INTERFACE I_Serializer EXTENDS I_Disposable

METHOD PUBLIC AddBase64 : I_Serializer
VAR_INPUT
	pBytes : POINTER TO BYTE;
	nBytes : DINT;
END_VAR
END_METHOD

METHOD PUBLIC AddBool : I_Serializer
VAR_INPUT
	Value : BOOL;
END_VAR
END_METHOD

METHOD PUBLIC AddByte : I_Serializer
VAR_INPUT
	Value : BYTE;
END_VAR
END_METHOD

METHOD PUBLIC AddBytesAsHex : I_Serializer
VAR_INPUT
	pBytes : POINTER TO BYTE;
	nBytes : DINT;
END_VAR
END_METHOD

METHOD PUBLIC AddDateTime : I_Serializer
VAR_INPUT
	Value : DATE_AND_TIME;
END_VAR
END_METHOD

METHOD PUBLIC AddDcTime : I_Serializer
VAR_INPUT
	Value : DCTIME;
END_VAR
END_METHOD

METHOD PUBLIC AddDint : I_Serializer
VAR_INPUT
	Value : DINT;
END_VAR
END_METHOD

METHOD PUBLIC AddDword : I_Serializer
VAR_INPUT
	Value : DWORD;
END_VAR
END_METHOD

METHOD PUBLIC AddFileTime : I_Serializer
VAR_INPUT
	Value : FILETIME;
END_VAR
END_METHOD

METHOD PUBLIC AddInt : I_Serializer
VAR_INPUT
	Value : INT;
END_VAR
END_METHOD

METHOD PUBLIC AddKey : I_Serializer
VAR_INPUT
	Key : T_MAXSTRING;
END_VAR
END_METHOD

METHOD PUBLIC AddKeyBase64 : I_Serializer
VAR_INPUT
	Key : T_MAXSTRING;
	pBytes : POINTER TO BYTE;
	nBytes : DINT;
END_VAR
END_METHOD

METHOD PUBLIC AddKeyBool : I_Serializer
VAR_INPUT
	Key : T_MAXSTRING;
	Value : BOOL;
END_VAR
END_METHOD

METHOD PUBLIC AddKeyByte : I_Serializer
VAR_INPUT
	Key : T_MAXSTRING;
	Value : BYTE;
END_VAR
END_METHOD

METHOD PUBLIC AddKeyBytesAsHex : I_Serializer
VAR_INPUT
	Key : T_MAXSTRING;
	pBytes : POINTER TO BYTE;
	nBytes : DINT;
END_VAR
END_METHOD

METHOD PUBLIC AddKeyDateTime : I_Serializer
VAR_INPUT
	Key : T_MAXSTRING;
	Value : DATE_AND_TIME;
END_VAR
END_METHOD

METHOD PUBLIC AddKeyDcTime : I_Serializer
VAR_INPUT
	Key : T_MAXSTRING;
	Value : DCTIME;
END_VAR
END_METHOD

METHOD PUBLIC AddKeyDint : I_Serializer
VAR_INPUT
	Key : T_MAXSTRING;
	Value : DINT;
END_VAR
END_METHOD

METHOD PUBLIC AddKeyDword : I_Serializer
VAR_INPUT
	Key : T_MAXSTRING;
	Value : DWORD;
END_VAR
END_METHOD

METHOD PUBLIC AddKeyFileTime : I_Serializer
VAR_INPUT
	Key : T_MAXSTRING;
	Value : FILETIME;
END_VAR
END_METHOD

METHOD PUBLIC AddKeyInt : I_Serializer
VAR_INPUT
	Key : T_MAXSTRING;
	Value : INT;
END_VAR
END_METHOD

METHOD PUBLIC AddKeyLint : I_Serializer
VAR_INPUT
	Key : T_MAXSTRING;
	Value : LINT;
END_VAR
END_METHOD

METHOD PUBLIC AddKeyLreal : I_Serializer
VAR_INPUT
	Key : T_MAXSTRING;
	Value : LREAL;
END_VAR
END_METHOD

METHOD PUBLIC AddKeyLtime : I_Serializer
VAR_INPUT
	Key : T_MAXSTRING;
	Value : LTIME;
END_VAR
END_METHOD

METHOD PUBLIC AddKeyLword : I_Serializer
VAR_INPUT
	Key : T_MAXSTRING;
	Value : LWORD;
END_VAR
END_METHOD

METHOD PUBLIC AddKeyNull : I_Serializer
VAR_INPUT
	Key : T_MAXSTRING;
END_VAR
END_METHOD

METHOD PUBLIC AddKeyReal : I_Serializer
VAR_INPUT
	Key : T_MAXSTRING;
	Value : REAL;
END_VAR
END_METHOD

METHOD PUBLIC AddKeySint : I_Serializer
VAR_INPUT
	Key : T_MAXSTRING;
	Value : SINT;
END_VAR
END_METHOD

METHOD PUBLIC AddKeyString : I_Serializer
VAR_INPUT
	Key : T_MAXSTRING;
	Value : T_MAXSTRING;
END_VAR
END_METHOD

METHOD PUBLIC AddKeyStringByRef : I_Serializer
VAR_INPUT
	Key : T_MAXSTRING;
	Value : REFERENCE TO STRING;
END_VAR
END_METHOD

METHOD PUBLIC AddKeyTime : I_Serializer
VAR_INPUT
	Key : T_MAXSTRING;
	Value : TIME;
END_VAR
END_METHOD

METHOD PUBLIC AddKeyTod : I_Serializer
VAR_INPUT
	Key : T_MAXSTRING;
	Value : TOD;
END_VAR
END_METHOD

METHOD PUBLIC AddKeyUdint : I_Serializer
VAR_INPUT
	Key : T_MAXSTRING;
	Value : UDINT;
END_VAR
END_METHOD

METHOD PUBLIC AddKeyUint : I_Serializer
VAR_INPUT
	Key : T_MAXSTRING;
	Value : UINT;
END_VAR
END_METHOD

METHOD PUBLIC AddKeyUlint : I_Serializer
VAR_INPUT
	Key : T_MAXSTRING;
	Value : ULINT;
END_VAR
END_METHOD

METHOD PUBLIC AddKeyUsint : I_Serializer
VAR_INPUT
	Key : T_MAXSTRING;
	Value : USINT;
END_VAR
END_METHOD

METHOD PUBLIC AddKeyWord : I_Serializer
VAR_INPUT
	Key : T_MAXSTRING;
	Value : WORD;
END_VAR
END_METHOD

METHOD PUBLIC AddLint : I_Serializer
VAR_INPUT
	Value : LINT;
END_VAR
END_METHOD

METHOD PUBLIC AddLreal : I_Serializer
VAR_INPUT
	Value : LREAL;
END_VAR
END_METHOD

METHOD PUBLIC AddLtime : I_Serializer
VAR_INPUT
	Value : LTIME;
END_VAR
END_METHOD

METHOD PUBLIC AddLword : I_Serializer
VAR_INPUT
	Value : LWORD;
END_VAR
END_METHOD

METHOD PUBLIC AddNull : I_Serializer
VAR_INPUT
END_VAR
END_METHOD

METHOD PUBLIC AddReal : I_Serializer
VAR_INPUT
	Value : REAL;
END_VAR
END_METHOD

METHOD PUBLIC AddSint : I_Serializer
VAR_INPUT
	Value : SINT;
END_VAR
END_METHOD

METHOD PUBLIC AddString : I_Serializer
VAR_INPUT
	Value : T_MAXSTRING;
END_VAR
END_METHOD

METHOD PUBLIC AddStringByRef : I_Serializer
VAR_INPUT
	Value : REFERENCE TO STRING;
END_VAR
END_METHOD

METHOD PUBLIC AddTime : I_Serializer
VAR_INPUT
	Value : TIME;
END_VAR
END_METHOD

METHOD PUBLIC AddTod : I_Serializer
VAR_INPUT
	Value : TOD;
END_VAR
END_METHOD

METHOD PUBLIC AddUdint : I_Serializer
VAR_INPUT
	Value : UDINT;
END_VAR
END_METHOD

METHOD PUBLIC AddUint : I_Serializer
VAR_INPUT
	Value : UINT;
END_VAR
END_METHOD

METHOD PUBLIC AddUlint : I_Serializer
VAR_INPUT
	Value : ULINT;
END_VAR
END_METHOD

METHOD PUBLIC AddUsint : I_Serializer
VAR_INPUT
	Value : USINT;
END_VAR
END_METHOD

METHOD PUBLIC AddWord : I_Serializer
VAR_INPUT
	Value : WORD;
END_VAR
END_METHOD

METHOD PUBLIC Clone : I_Serializer
END_METHOD

METHOD PUBLIC EndArray : I_Serializer
VAR_INPUT
END_VAR
END_METHOD

METHOD PUBLIC EndObject : I_Serializer
VAR_INPUT
END_VAR
END_METHOD

METHOD PUBLIC GetSeralizedDataLength : UDINT
VAR_INPUT
END_VAR
END_METHOD

METHOD PUBLIC Reset
VAR_INPUT
END_VAR
END_METHOD

METHOD PUBLIC StartArray : I_Serializer
VAR_INPUT
END_VAR
END_METHOD

METHOD PUBLIC StartObject : I_Serializer
VAR_INPUT
END_VAR
END_METHOD

METHOD TryCopySerialziedData : BOOL
VAR_INPUT
	DestinationAddress : PVOID;
	DestinationSize : UDINT;
END_VAR
END_METHOD

METHOD TryGetSerialziedData : BOOL
VAR_INPUT
	DestinationAddress : PVOID;
	DestinationSize : UDINT;
END_VAR
END_METHOD

END_INTERFACE

(* stored: Version 1.1.0.1, ProductVersion 3.1.4024.12
   Itf I_Serializer: Id {1915cd37-a63c-497b-b451-ce60404fe3d9}
   Method AddBase64: Id {9a2f81bf-aaf2-40ff-bc78-2f248fef6daf}
   Method AddBool: Id {7c9eb409-6a97-464c-b9e8-37bd91ca50e0}
   Method AddByte: Id {9c7da6f3-c934-058b-3f86-fbbe37b50c50}
   Method AddBytesAsHex: Id {feb24363-968e-412e-a13a-58f511bce576}
   Method AddDateTime: Id {787ca0f0-ca02-4323-991c-1e163a2b8af9}
   Method AddDcTime: Id {96c51290-7094-42a8-be20-9fb3a4d0bac9}
   Method AddDint: Id {995f0327-1ab2-4c65-a0b3-c5d955682216}
   Method AddDword: Id {cc56a495-91d4-0ddb-1546-d72f711986c2}
   Method AddFileTime: Id {489c5bc3-d184-4bca-a5f4-5c5f7f70baa2}
   Method AddInt: Id {2d6f4f5c-c8a8-034d-0498-846c1f9c03c1}
   Method AddKey: Id {7181a5f6-a406-435b-882f-40133bfca485}
   Method AddKeyBase64: Id {a2dc03fb-6ad8-4821-a6b8-a591e682e648}
   Method AddKeyBool: Id {0ad5b9aa-463d-44c4-b5b6-ea0ede55b5f0}
   Method AddKeyByte: Id {673c045a-084f-0fc8-06b3-07b336d49c45}
   Method AddKeyBytesAsHex: Id {dd3ce26e-aa72-46c8-a573-d46dbb58113d}
   Method AddKeyDateTime: Id {a4563e1e-0bb3-4f05-8877-05d1ba1631b6}
   Method AddKeyDcTime: Id {fb1ffde4-5fdb-4c8a-b8a7-5b40a265de64}
   Method AddKeyDint: Id {2203b447-9d10-45e2-9579-df0fefa39614}
   Method AddKeyDword: Id {b2befd78-8d14-041f-07b5-5e9bd962bd6a}
   Method AddKeyFileTime: Id {5b348315-e1a8-4262-a189-a25825ec5c35}
   Method AddKeyInt: Id {58637fe8-d6bd-0e9a-13f0-5862d6b7a036}
   Method AddKeyLint: Id {94e7f731-3ca6-4d76-88d4-f5a73d926b38}
   Method AddKeyLreal: Id {903b30b2-c389-4ce1-af78-2064041a9245}
   Method AddKeyLtime: Id {a56856e3-4877-0dc0-38ad-7742e0167ea6}
   Method AddKeyLword: Id {10bfb51b-a5fb-029d-33e0-f59b87248184}
   Method AddKeyNull: Id {cf4e9ea8-4550-47d2-b465-e0d85e4b7ed8}
   Method AddKeyReal: Id {dd8ea360-144c-42c7-a4e1-38913b192e00}
   Method AddKeySint: Id {ce53949b-54f8-0014-1a41-d6640e10a99d}
   Method AddKeyString: Id {b377c3c4-7ad1-0539-3da9-cf2f74ba9cfa}
   Method AddKeyStringByRef: Id {aa12f636-cd25-4eeb-a6d4-5c98d2326d61}
   Method AddKeyTime: Id {fe3dee30-5f6e-0d6f-0c7f-4f821dd9fe03}
   Method AddKeyTod: Id {c1df6a10-99e1-0661-2303-5e9bb0a0e03d}
   Method AddKeyUdint: Id {454ef19f-e877-4afb-9896-2c6339e62e98}
   Method AddKeyUint: Id {9bc1a8b9-8875-043d-2651-15cbe1e038f9}
   Method AddKeyUlint: Id {753d5520-149b-41ab-aadc-4c0b7d4dbd6e}
   Method AddKeyUsint: Id {706177a6-afb0-0138-32fc-e76a12fea32d}
   Method AddKeyWord: Id {0618121c-f73f-0667-086a-2bafa3f64b4c}
   Method AddLint: Id {6ff67be4-be94-46e1-9ef6-9a3b60a3f24a}
   Method AddLreal: Id {ae7879ac-f834-4469-b087-debf704489d2}
   Method AddLtime: Id {677a15ab-9040-022e-0d00-47c08cb1124a}
   Method AddLword: Id {56ebdd15-26ed-0ece-30b5-305b24bd6747}
   Method AddNull: Id {0ce856e1-0d16-4254-943c-9d399b151f53}
   Method AddReal: Id {37a1ed66-5e4c-49c9-a63a-d06d4077642d}
   Method AddSint: Id {7781586a-f051-045d-3200-1a531d3be826}
   Method AddString: Id {97868ca8-e46c-0736-2cfd-d37ea6cabe3c}
   Method AddStringByRef: Id {f2264a10-2f67-4248-a367-daf32bea1d9f}
   Method AddTime: Id {0d2f9377-10ee-0af4-3e45-af5ad44dba64}
   Method AddTod: Id {64a90bf0-1955-0fd0-12ea-a7a4b297542c}
   Method AddUdint: Id {24c09bd3-0ea6-460d-bb0e-5cc5f70b11be}
   Method AddUint: Id {f6301b62-2ac9-0962-3e2a-ced01a95c7f1}
   Method AddUlint: Id {01563e0f-9fc7-4275-8bd4-f1b12ec84106}
   Method AddUsint: Id {b5b679bb-0f72-0718-099d-142957f977ab}
   Method AddWord: Id {21a5be39-aabe-07c2-1eed-342a3a0701f4}
   Method Clone: Id {03335a3b-3001-4635-98a3-93c6b3d47142}
   Method EndArray: Id {608e5786-8bdc-4b9e-8097-ef16e4371389}
   Method EndObject: Id {0ed3b762-d376-451a-bfd4-b47bfa7de97c}
   Method GetSeralizedDataLength: Id {dd25f96d-06dc-4960-8c8c-b867ac96101a}
   Method Reset: Id {75b14756-7d52-4511-9104-dc66d7f097ec}
   Method StartArray: Id {8ef4260f-1a7f-455b-854a-0bfd72820fa8}
   Method StartObject: Id {f5ce7294-a584-4d95-878b-0aaddb33692e}
   Method TryCopySerialziedData: Id {b089a511-aa82-4ea4-a966-f29e05751c4c}
   Method TryGetSerialziedData: Id {f7ffa1bd-a3ef-402a-8560-d7216b36be70} *)
